PROGRAM popup
VAR
	fbOpenMessageDialogEmergency: R_trig;
END_VAR

fbOpenMessageDialogEmergency(CLK := gvl.emergency);
IF fbOpenMessageDialogEmergency.Q  THEN
	OpenMessageDialogEmergency();
END_IF

END_PROGRAM

(* stored: Version 1.1.0.1, ProductVersion 3.1.4024.12
   POU popup: Id {5414fea7-f943-44c1-9c82-35278987b2fa}, SpecialFunc None *)
